FUNCTION_BLOCK InputPort_Trigger EXTENDS InputPort implements I_TriggerPort
VAR
END_VAR

PROPERTY PUBLIC Result : HRESULT
GET
VAR
	hresult : HRESULT;
END_VAR
TryGet(hresult);
Result := hresult;
END_GET
END_PROPERTY

END_FUNCTION_BLOCK

(* stored: Version 1.1.0.1, ProductVersion 3.1.4024.12
   POU InputPort_Trigger: Id {c02d3224-6f96-0f96-1fe9-600e6363abf5}, SpecialFunc None
   Property Result: Id {e576605c-d71f-09ed-3b63-61daa81508ae}
   Get Get: Id {b83faf8c-762a-07b7-167e-c1a16ae1bf48} *)
